// Mitsubishi GX Works2 project: b2   PLC: Q03UDE

// global labels: Global1
VAR_GLOBAL
  startstop AT X40 : BOOL;
  estopbt AT X41 : BOOL;
  thuanbt AT X42 : BOOL;
  nguocbt AT X43 : BOOL;
  qt AT Y50 : BOOL;
  qn AT Y51 : BOOL;
END_VAR

PROGRAM MAIN
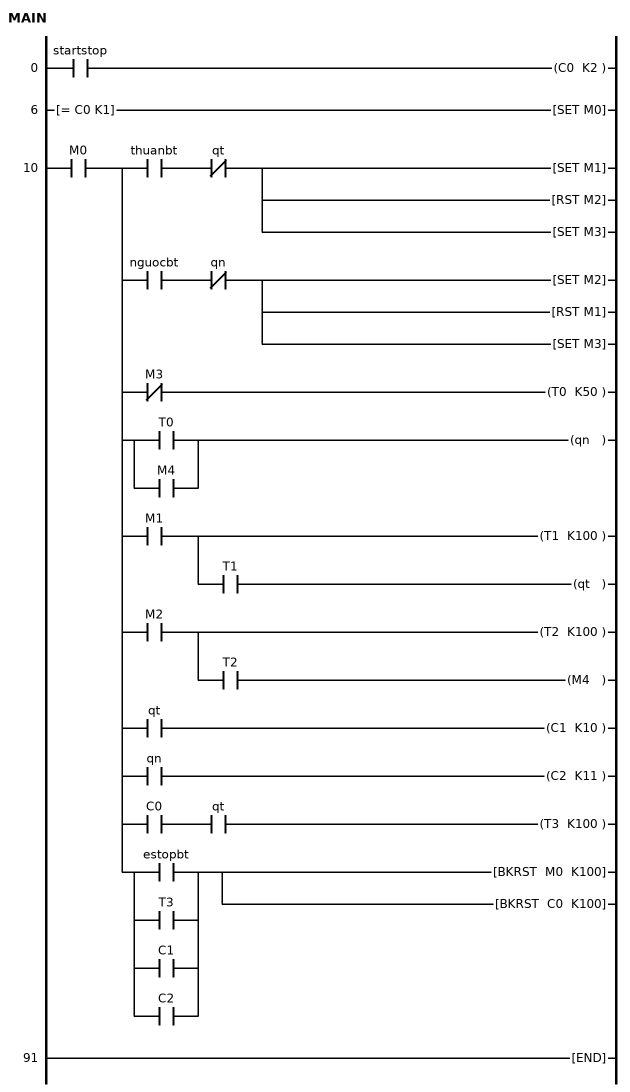
0     LD      startstop
      OUT     C0 K2
6     LD=     C0 K1
      SET     M0
10    LD      M0
      MPS
      AND     thuanbt
      ANI     qt
      SET     M1
      RST     M2
      SET     M3
      MRD
      AND     nguocbt
      ANI     qn
      SET     M2
      RST     M1
      SET     M3
      MRD
      ANI     M3
      OUT     T0 K50
      MRD
      LD      T0
      OR      M4
      ANB
      OUT     qn
      MRD
      AND     M1
      OUT     T1 K100
      AND     T1
      OUT     qt
      MRD
      AND     M2
      OUT     T2 K100
      AND     T2
      OUT     M4
      MRD
      AND     qt
      OUT     C1 K10
      MRD
      AND     qn
      OUT     C2 K11
      MRD
      AND     C0
      AND     qt
      OUT     T3 K100
      MPP
      LD      estopbt
      OR      T3
      OR      C1
      OR      C2
      ANB
      BKRST   M0 K100
      BKRST   C0 K100
91    END
END_PROGRAM
